(* Logix 5000 project; controller Project1Template vendor 1 type 14 code 151 rev 33.12; software revision 33.01; part 2 of 2 *)
(* tags used below, declared in another part *)
   SIM_ClampA : AOI_SIM_2PosCyl_ExtRet;
   SIM_ClampB : AOI_SIM_2PosCyl_ExtRet;
   SIM_ClampC : AOI_SIM_2PosCyl_ExtRet;
   SIM_EmptyFixture : TIMER;
   SIM_Fasten1 : AOI_SIM_RandomDelay;
   SIM_Fasten2 : AOI_SIM_RandomDelay;
   SIM_Fasten3 : AOI_SIM_RandomDelay;
   SIM_Fasten4 : AOI_SIM_RandomDelay;
   SIM_Fixture : AOI_SIM_2PosCyl_ExtRet;
   SIM_LightCurtainPartPlace : AOI_SIM_RandomDelay;
   SIM_LightCurtainPartRem : AOI_SIM_RandomDelay;
   SIM_NOP : BOOL;
   SIM_Oneshots : DINT;
   SIM_OperatorWorking : AOI_SIM_RandomDelay;
   SIM_PP_OFF : AOI_SIM_RandomDelay;
   SIM_PPA_ON : AOI_SIM_RandomDelay;
   SIM_PPB_ON : AOI_SIM_RandomDelay;
   SIM_PPC_ON : AOI_SIM_RandomDelay;
   SIM_PPD_ON : AOI_SIM_RandomDelay;
   SIM_RobotClear : AOI_SIM_RandomDelay;
   SIM_Torque : AOI_SIMAnalogSensor;
   F1_PASS : COUNTER;
   F2_PASS : COUNTER;
   F3_PASS : COUNTER;
   F4_PASS : COUNTER;
   FASTEN_AllComplete : BOOL;
   FASTEN_AllTorquesFail : BOOL;
   FASTEN_AllTorquesPass : BOOL;
   FASTEN_F1Complete : BOOL;
   FASTEN_F1Complete_ONS : BOOL;
   FASTEN_F1Torque : REAL;
   FASTEN_F1TorqueFail : BOOL;
   FASTEN_F1TorquePass : BOOL;
   FASTEN_F2Complete : BOOL;
   FASTEN_F2Complete_ONS : BOOL;
   FASTEN_F2Torque : REAL;
   FASTEN_F2TorqueFail : BOOL;
   FASTEN_F2TorquePass : BOOL;
   FASTEN_F3Complete : BOOL;
   FASTEN_F3Complete_ONS : BOOL;
   FASTEN_F3Torque : REAL;
   FASTEN_F3TorqueFail : BOOL;
   FASTEN_F3TorquePass : BOOL;
   FASTEN_F4Complete : BOOL;
   FASTEN_F4Complete_ONS : BOOL;
   FASTEN_F4Torque : REAL;
   FASTEN_F4TorqueFail : BOOL;
   FASTEN_F4TorquePass : BOOL;
   FASTEN_TorqueFeedback : REAL;
   FAULTS : DINT;
   FIXTURE_AllPartsPresent : BOOL;
   FIXTURE_AtHomePos : BOOL;
   FIXTURE_Empty : BOOL;
   FIXTURE_PartsSecured : BOOL;
   FIXTURE_PartsSecuredTmr : TIMER;
   FromHMI_ExtClampA_PB : BOOL;
   FromHMI_ExtClampB_PB : BOOL;
   FromHMI_ExtClampC_PB : BOOL;
   FromHMI_ExtFixture_PB : BOOL;
   FromHMI_F1LowLim : REAL;
   FromHMI_F1UppLim : REAL;
   FromHMI_F2LowLim : REAL;
   FromHMI_F2UppLim : REAL;
   FromHMI_F3LowLim : REAL;
   FromHMI_F3UppLim : REAL;
   FromHMI_F4LowLim : REAL;
   FromHMI_F4UppLim : REAL;
   FromHMI_RetClampA_PB : BOOL;
   FromHMI_RetClampB_PB : BOOL;
   FromHMI_RetClampC_PB : BOOL;
   FromHMI_RetFixture_PB : BOOL;
   FromHMI_StartPB : BOOL;
   FromHMI_StopPB : BOOL;
   FromRbt_ClearOfFixture : BOOL;
   FromRbt_Fasten1Complete : BOOL;
   FromRbt_Fasten2Complete : BOOL;
   FromRbt_Fasten3Complete : BOOL;
   FromRbt_Fasten4Complete : BOOL;
   HomePB : BOOL;
   I1 : INT;
   I2_CHA : REAL;   // Torque Sensor Input
   O3 : INT;
   SYS_AutoModeActive : BOOL;
   SYS_CycleActive : BOOL;
   SYS_ManualModeActive : BOOL;
   SYS_StartPBPulseTmr : TIMER;
   TIME : REAL;
   ToRbt_Fasten1Start : BOOL;
   ToRbt_Fasten2Start : BOOL;
   ToRbt_Fasten3Start : BOOL;
   ToRbt_Fasten4Start : BOOL;
(* MainProgram, continued *)

ROUTINE MainRoutine   (* ladder *)
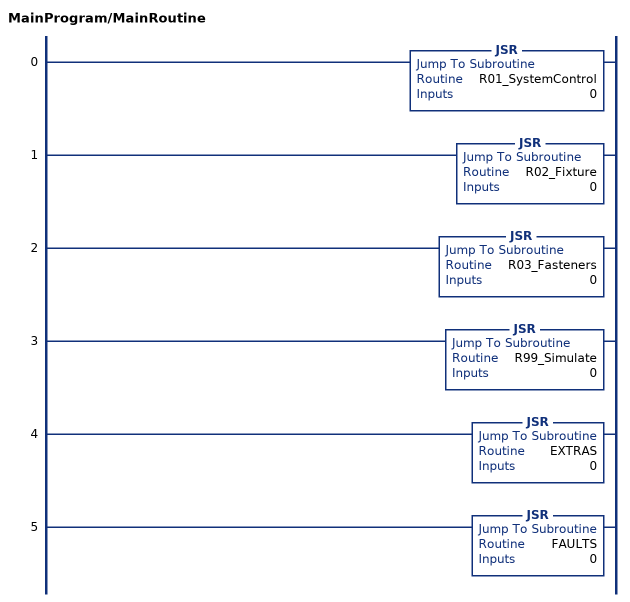
   0: JSR(R01_SystemControl,0);
   1: JSR(R02_Fixture,0);
   2: JSR(R03_Fasteners,0);
   3: JSR(R99_Simulate,0);
   4: JSR(EXTRAS,0);
   5: JSR(FAULTS,0);
END_ROUTINE

ROUTINE R01_SystemControl   (* ladder *)
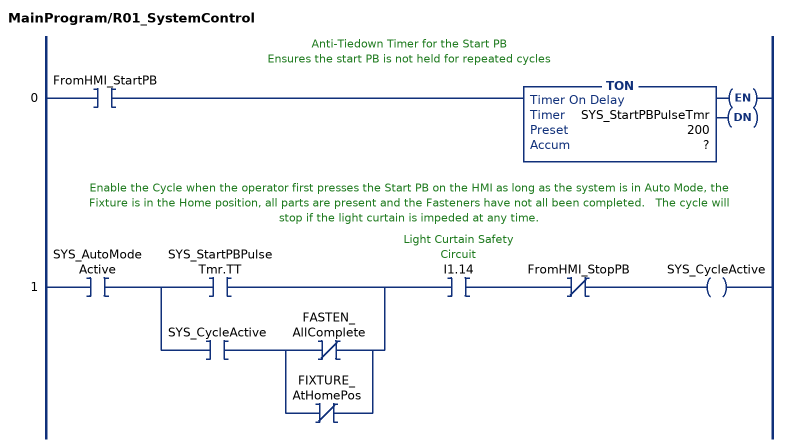
   // Anti-Tiedown Timer for the Start PB
   // Ensures the start PB is not held for repeated cycles
   0: XIC(FromHMI_StartPB)TON(SYS_StartPBPulseTmr,?,?);
   // Enable the Cycle when the operator first presses the Start PB on the HMI as long as the system is in Auto Mode, the Fixture is in the Home position, all parts are present and the Fasteners have not all been completed.   The cycle will stop if the light curtain is impeded at any time.
   1: XIC(SYS_AutoModeActive)[XIC(SYS_StartPBPulseTmr.TT) ,XIC(SYS_CycleActive) [XIO(FASTEN_AllComplete) ,XIO(FIXTURE_AtHomePos) ] ]XIC(I1.14)XIO(FromHMI_StopPB)OTE(SYS_CycleActive);
END_ROUTINE

ROUTINE R02_Fixture   (* ladder *)
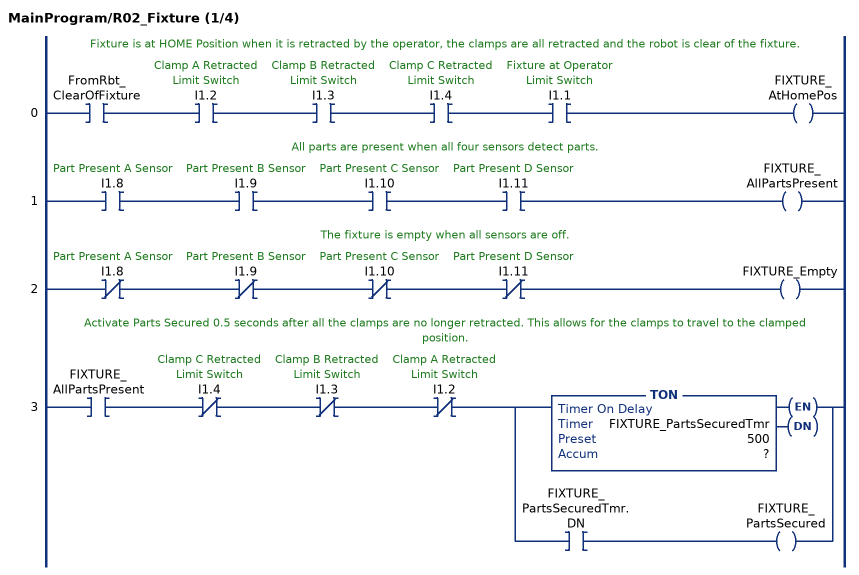
   // Fixture is at HOME Position when it is retracted by the operator, the clamps are all retracted and the robot is clear of the fixture.
   0: XIC(FromRbt_ClearOfFixture)XIC(I1.2)XIC(I1.3)XIC(I1.4)XIC(I1.1)OTE(FIXTURE_AtHomePos);
   // All parts are present when all four sensors detect parts.
   1: XIC(I1.8)XIC(I1.9)XIC(I1.10)XIC(I1.11)OTE(FIXTURE_AllPartsPresent);
   // The fixture is empty when all sensors are off.
   2: XIO(I1.8)XIO(I1.9)XIO(I1.10)XIO(I1.11)OTE(FIXTURE_Empty);
   // Activate Parts Secured 0.5 seconds after all the clamps are no longer retracted. This allows for the clamps to travel to the clamped position.
   3: XIC(FIXTURE_AllPartsPresent)XIO(I1.4)XIO(I1.3)XIO(I1.2)[TON(FIXTURE_PartsSecuredTmr,?,?) ,XIC(FIXTURE_PartsSecuredTmr.DN) OTE(FIXTURE_PartsSecured) ];
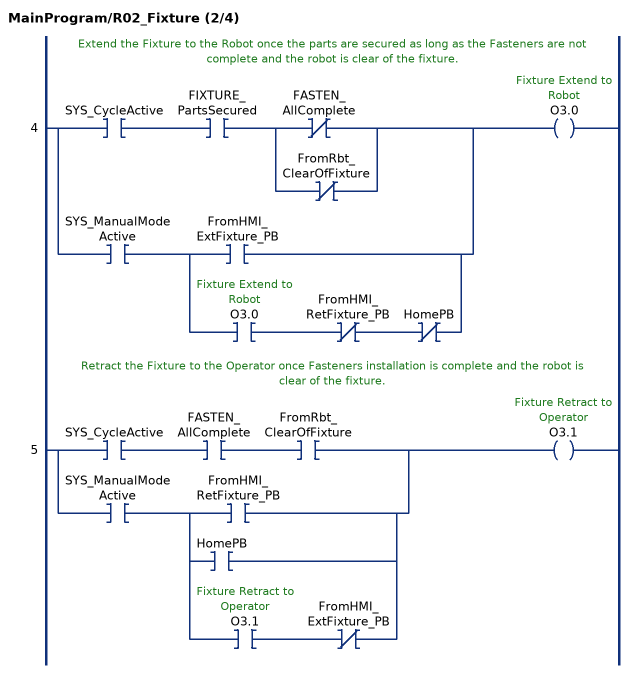
   // Extend the Fixture to the Robot once the parts are secured as long as the Fasteners are not complete and the robot is clear of the fixture.
   4: [XIC(SYS_CycleActive) XIC(FIXTURE_PartsSecured) [XIO(FASTEN_AllComplete) ,XIO(FromRbt_ClearOfFixture) ] ,XIC(SYS_ManualModeActive) [XIC(FromHMI_ExtFixture_PB) ,XIC(O3.0) XIO(FromHMI_RetFixture_PB) XIO(HomePB) ] ]OTE(O3.0);
   // Retract the Fixture to the Operator once Fasteners installation is complete and the robot is clear of the fixture.
   5: [XIC(SYS_CycleActive) XIC(FASTEN_AllComplete) XIC(FromRbt_ClearOfFixture) ,XIC(SYS_ManualModeActive) [[XIC(FromHMI_RetFixture_PB) ,XIC(HomePB) ] ,XIC(O3.1) XIO(FromHMI_ExtFixture_PB) ] ]OTE(O3.1);
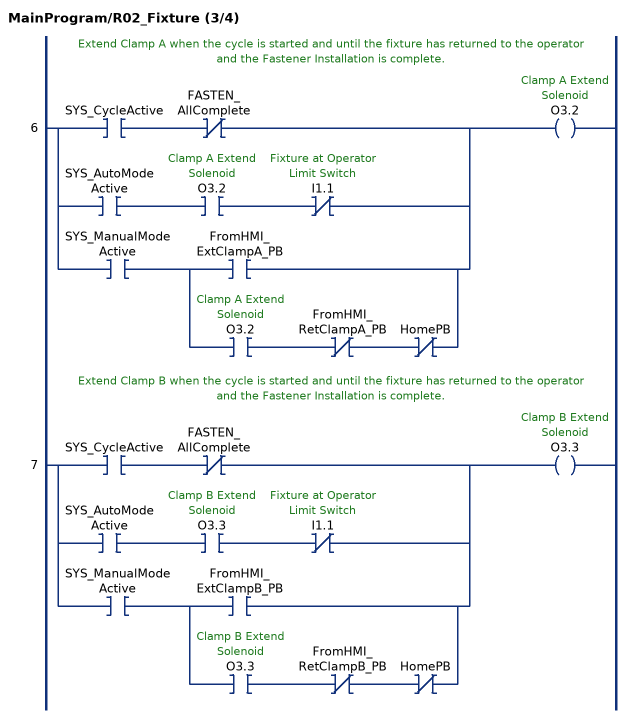
   // Extend Clamp A when the cycle is started and until the fixture has returned to the operator and the Fastener Installation is complete.
   6: [XIC(SYS_CycleActive) XIO(FASTEN_AllComplete) ,XIC(SYS_AutoModeActive) XIC(O3.2) XIO(I1.1) ,XIC(SYS_ManualModeActive) [XIC(FromHMI_ExtClampA_PB) ,XIC(O3.2) XIO(FromHMI_RetClampA_PB) XIO(HomePB) ] ]OTE(O3.2);
   // Extend Clamp B when the cycle is started and until the fixture has returned to the operator and the Fastener Installation is complete.
   7: [XIC(SYS_CycleActive) XIO(FASTEN_AllComplete) ,XIC(SYS_AutoModeActive) XIC(O3.3) XIO(I1.1) ,XIC(SYS_ManualModeActive) [XIC(FromHMI_ExtClampB_PB) ,XIC(O3.3) XIO(FromHMI_RetClampB_PB) XIO(HomePB) ] ]OTE(O3.3);
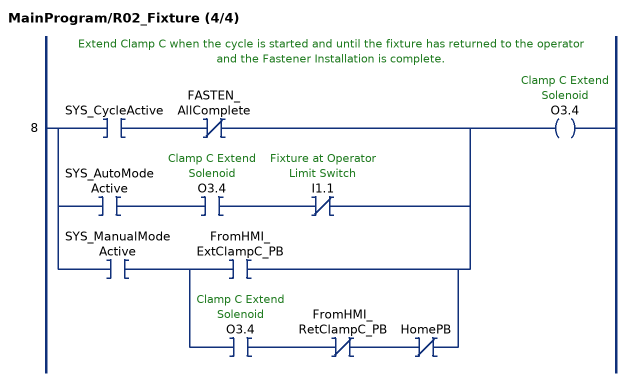
   // Extend Clamp C when the cycle is started and until the fixture has returned to the operator and the Fastener Installation is complete.
   8: [XIC(SYS_CycleActive) XIO(FASTEN_AllComplete) ,XIC(SYS_AutoModeActive) XIC(O3.4) XIO(I1.1) ,XIC(SYS_ManualModeActive) [XIC(FromHMI_ExtClampC_PB) ,XIC(O3.4) XIO(FromHMI_RetClampC_PB) XIO(HomePB) ] ]OTE(O3.4);
END_ROUTINE

ROUTINE R03_Fasteners   (* ladder *)
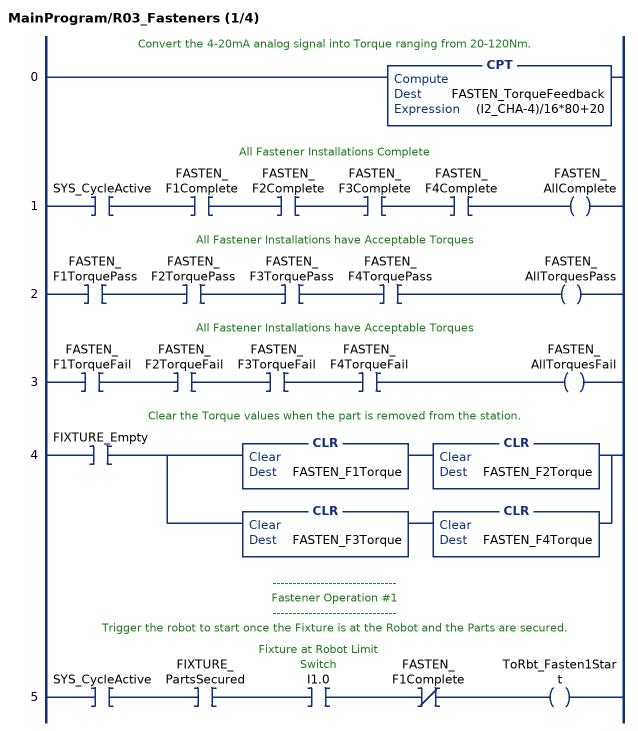
   // Convert the 4-20mA analog signal into Torque ranging from 20-120Nm.
   0: CPT(FASTEN_TorqueFeedback,(I2_CHA-4)/16*80+20);
   // All Fastener Installations Complete
   1: XIC(SYS_CycleActive)XIC(FASTEN_F1Complete)XIC(FASTEN_F2Complete)XIC(FASTEN_F3Complete)XIC(FASTEN_F4Complete)OTE(FASTEN_AllComplete);
   // All Fastener Installations have Acceptable Torques
   2: XIC(FASTEN_F1TorquePass)XIC(FASTEN_F2TorquePass)XIC(FASTEN_F3TorquePass)XIC(FASTEN_F4TorquePass)OTE(FASTEN_AllTorquesPass);
   // All Fastener Installations have Acceptable Torques
   3: XIC(FASTEN_F1TorqueFail)XIC(FASTEN_F2TorqueFail)XIC(FASTEN_F3TorqueFail)XIC(FASTEN_F4TorqueFail)OTE(FASTEN_AllTorquesFail);
   // Clear the Torque values when the part is removed from the station.
   4: XIC(FIXTURE_Empty)[CLR(FASTEN_F1Torque) CLR(FASTEN_F2Torque) ,CLR(FASTEN_F3Torque) CLR(FASTEN_F4Torque) ];
   // -------------------------------
   // Fastener Operation #1
   // -------------------------------
   // Trigger the robot to start once the Fixture is at the Robot and the Parts are secured.
   5: XIC(SYS_CycleActive)XIC(FIXTURE_PartsSecured)XIC(I1.0)XIO(FASTEN_F1Complete)OTE(ToRbt_Fasten1Start);
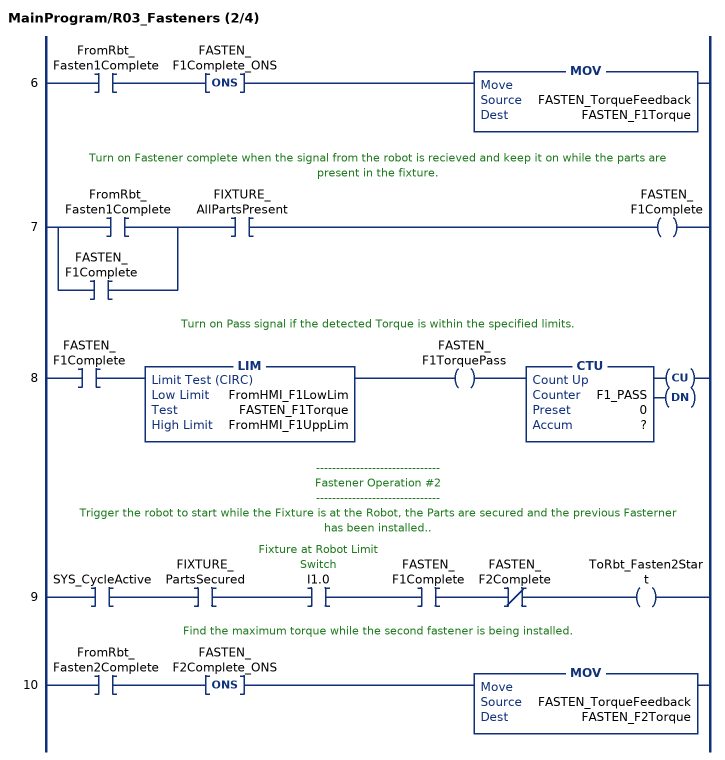
   6: XIC(FromRbt_Fasten1Complete)ONS(FASTEN_F1Complete_ONS)MOV(FASTEN_TorqueFeedback,FASTEN_F1Torque);
   // Turn on Fastener complete when the signal from the robot is recieved and keep it on while the parts are present in the fixture.
   7: [XIC(FromRbt_Fasten1Complete) ,XIC(FASTEN_F1Complete) ]XIC(FIXTURE_AllPartsPresent)OTE(FASTEN_F1Complete);
   // Turn on Pass signal if the detected Torque is within the specified limits.
   8: XIC(FASTEN_F1Complete)LIM(FromHMI_F1LowLim,FASTEN_F1Torque,FromHMI_F1UppLim)OTE(FASTEN_F1TorquePass)CTU(F1_PASS,?,?);
   // -------------------------------
   // Fastener Operation #2
   // -------------------------------
   // Trigger the robot to start while the Fixture is at the Robot, the Parts are secured and the previous Fasterner has been installed..
   9: XIC(SYS_CycleActive)XIC(FIXTURE_PartsSecured)XIC(I1.0)XIC(FASTEN_F1Complete)XIO(FASTEN_F2Complete)OTE(ToRbt_Fasten2Start);
   // Find the maximum torque while the second fastener is being installed.
   10: XIC(FromRbt_Fasten2Complete)ONS(FASTEN_F2Complete_ONS)MOV(FASTEN_TorqueFeedback,FASTEN_F2Torque);
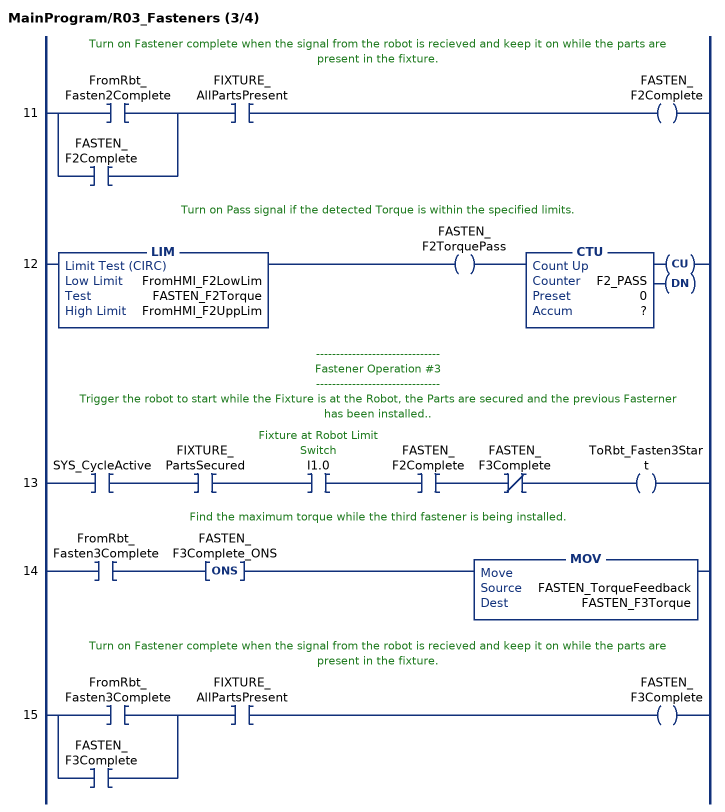
   // Turn on Fastener complete when the signal from the robot is recieved and keep it on while the parts are present in the fixture.
   11: [XIC(FromRbt_Fasten2Complete) ,XIC(FASTEN_F2Complete) ]XIC(FIXTURE_AllPartsPresent)OTE(FASTEN_F2Complete);
   // Turn on Pass signal if the detected Torque is within the specified limits.
   12: LIM(FromHMI_F2LowLim,FASTEN_F2Torque,FromHMI_F2UppLim)OTE(FASTEN_F2TorquePass)CTU(F2_PASS,?,?);
   // -------------------------------
   // Fastener Operation #3
   // -------------------------------
   // Trigger the robot to start while the Fixture is at the Robot, the Parts are secured and the previous Fasterner has been installed..
   13: XIC(SYS_CycleActive)XIC(FIXTURE_PartsSecured)XIC(I1.0)XIC(FASTEN_F2Complete)XIO(FASTEN_F3Complete)OTE(ToRbt_Fasten3Start);
   // Find the maximum torque while the third fastener is being installed.
   14: XIC(FromRbt_Fasten3Complete)ONS(FASTEN_F3Complete_ONS)MOV(FASTEN_TorqueFeedback,FASTEN_F3Torque);
   // Turn on Fastener complete when the signal from the robot is recieved and keep it on while the parts are present in the fixture.
   15: [XIC(FromRbt_Fasten3Complete) ,XIC(FASTEN_F3Complete) ]XIC(FIXTURE_AllPartsPresent)OTE(FASTEN_F3Complete);
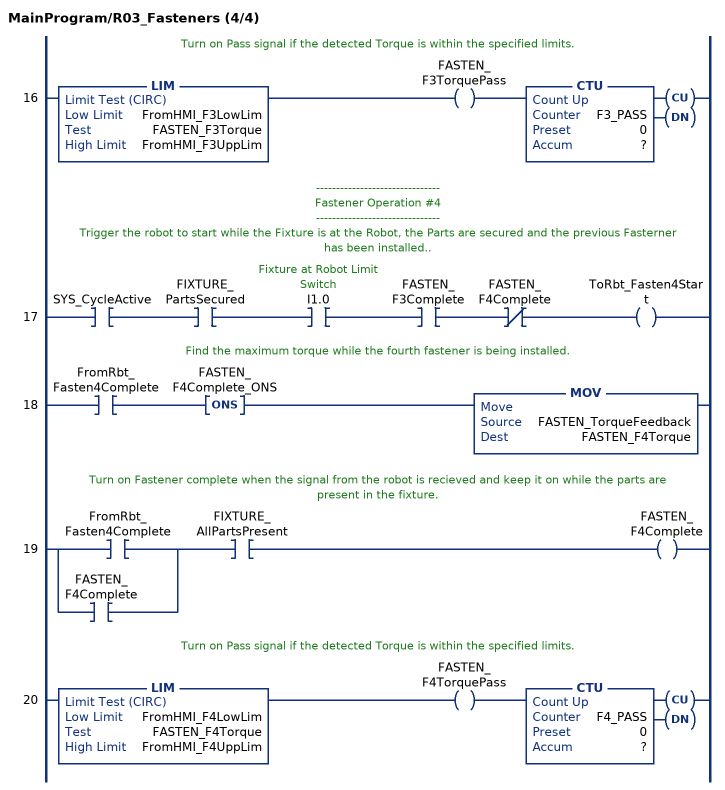
   // Turn on Pass signal if the detected Torque is within the specified limits.
   16: LIM(FromHMI_F3LowLim,FASTEN_F3Torque,FromHMI_F3UppLim)OTE(FASTEN_F3TorquePass)CTU(F3_PASS,?,?);
   // -------------------------------
   // Fastener Operation #4
   // -------------------------------
   // Trigger the robot to start while the Fixture is at the Robot, the Parts are secured and the previous Fasterner has been installed..
   17: XIC(SYS_CycleActive)XIC(FIXTURE_PartsSecured)XIC(I1.0)XIC(FASTEN_F3Complete)XIO(FASTEN_F4Complete)OTE(ToRbt_Fasten4Start);
   // Find the maximum torque while the fourth fastener is being installed.
   18: XIC(FromRbt_Fasten4Complete)ONS(FASTEN_F4Complete_ONS)MOV(FASTEN_TorqueFeedback,FASTEN_F4Torque);
   // Turn on Fastener complete when the signal from the robot is recieved and keep it on while the parts are present in the fixture.
   19: [XIC(FromRbt_Fasten4Complete) ,XIC(FASTEN_F4Complete) ]XIC(FIXTURE_AllPartsPresent)OTE(FASTEN_F4Complete);
   // Turn on Pass signal if the detected Torque is within the specified limits.
   20: LIM(FromHMI_F4LowLim,FASTEN_F4Torque,FromHMI_F4UppLim)OTE(FASTEN_F4TorquePass)CTU(F4_PASS,?,?);
END_ROUTINE

ROUTINE R98_DemoMonitoring   (* ladder *)
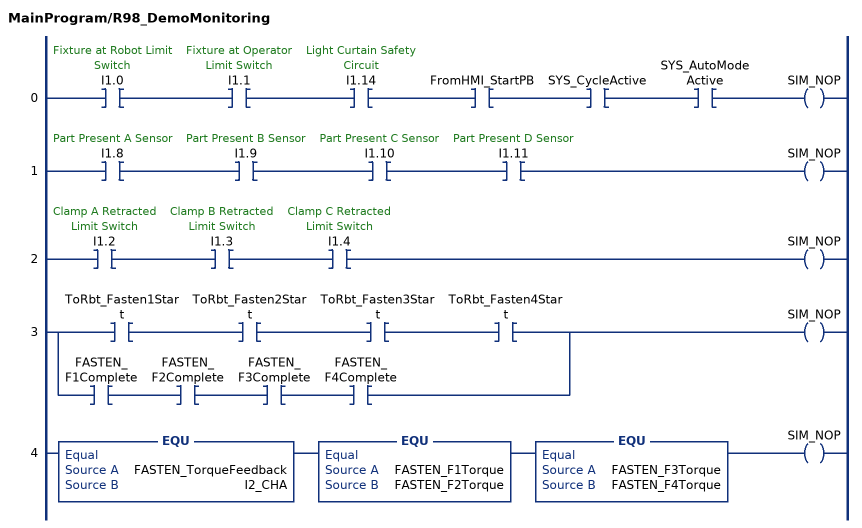
   0: XIC(I1.0)XIC(I1.1)XIC(I1.14)XIC(FromHMI_StartPB)XIC(SYS_CycleActive)XIC(SYS_AutoModeActive)OTE(SIM_NOP);
   1: XIC(I1.8)XIC(I1.9)XIC(I1.10)XIC(I1.11)OTE(SIM_NOP);
   2: XIC(I1.2)XIC(I1.3)XIC(I1.4)OTE(SIM_NOP);
   3: [XIC(ToRbt_Fasten1Start) XIC(ToRbt_Fasten2Start) XIC(ToRbt_Fasten3Start) XIC(ToRbt_Fasten4Start) ,XIC(FASTEN_F1Complete) XIC(FASTEN_F2Complete) XIC(FASTEN_F3Complete) XIC(FASTEN_F4Complete) ]OTE(SIM_NOP);
   4: EQU(FASTEN_TorqueFeedback,I2_CHA)EQU(FASTEN_F1Torque,FASTEN_F2Torque)EQU(FASTEN_F3Torque,FASTEN_F4Torque)OTE(SIM_NOP);
END_ROUTINE

ROUTINE R99_Simulate   (* ladder *)
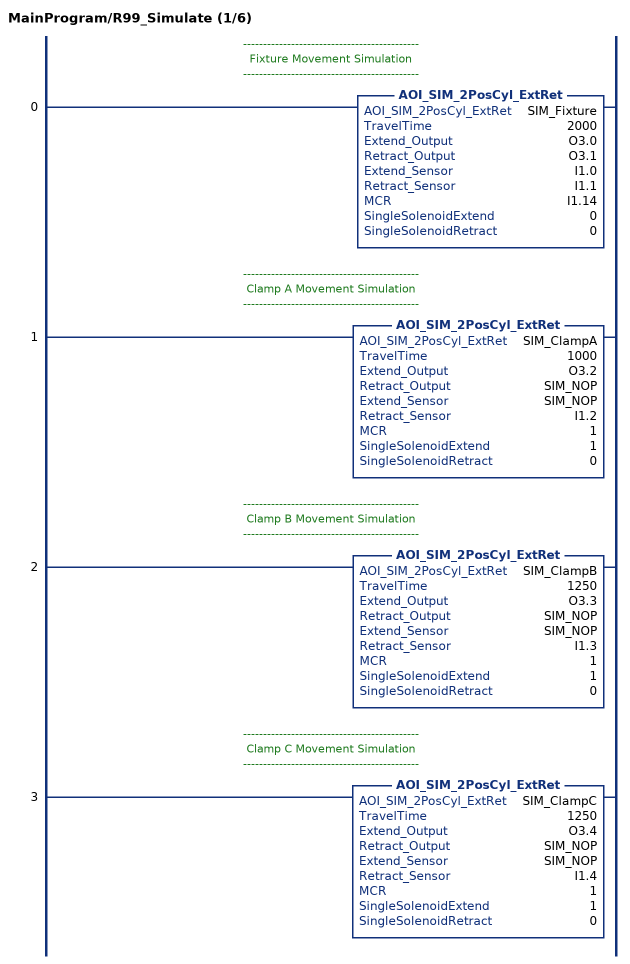
   // --------------------------------------------
   // Fixture Movement Simulation
   // --------------------------------------------
   0: AOI_SIM_2PosCyl_ExtRet(SIM_Fixture,2000,O3.0,O3.1,I1.0,I1.1,I1.14,0,0);
   // --------------------------------------------
   // Clamp A Movement Simulation
   // --------------------------------------------
   1: AOI_SIM_2PosCyl_ExtRet(SIM_ClampA,1000,O3.2,SIM_NOP,SIM_NOP,I1.2,1,1,0);
   // --------------------------------------------
   // Clamp B Movement Simulation
   // --------------------------------------------
   2: AOI_SIM_2PosCyl_ExtRet(SIM_ClampB,1250,O3.3,SIM_NOP,SIM_NOP,I1.3,1,1,0);
   // --------------------------------------------
   // Clamp C Movement Simulation
   // --------------------------------------------
   3: AOI_SIM_2PosCyl_ExtRet(SIM_ClampC,1250,O3.4,SIM_NOP,SIM_NOP,I1.4,1,1,0);
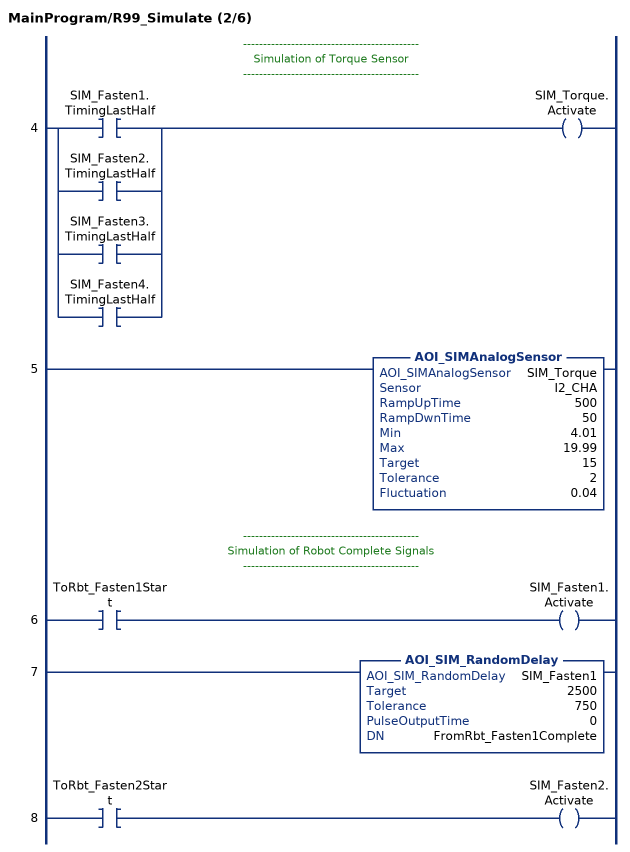
   // --------------------------------------------
   // Simulation of Torque Sensor
   // --------------------------------------------
   4: [XIC(SIM_Fasten1.TimingLastHalf) ,XIC(SIM_Fasten2.TimingLastHalf) ,XIC(SIM_Fasten3.TimingLastHalf) ,XIC(SIM_Fasten4.TimingLastHalf) ]OTE(SIM_Torque.Activate);
   5: AOI_SIMAnalogSensor(SIM_Torque,I2_CHA,500,50,4.01,19.99,15,2,0.04);
   // --------------------------------------------
   // Simulation of Robot Complete Signals
   // --------------------------------------------
   6: XIC(ToRbt_Fasten1Start)OTE(SIM_Fasten1.Activate);
   7: AOI_SIM_RandomDelay(SIM_Fasten1,2500,750,0,FromRbt_Fasten1Complete);
   8: XIC(ToRbt_Fasten2Start)OTE(SIM_Fasten2.Activate);
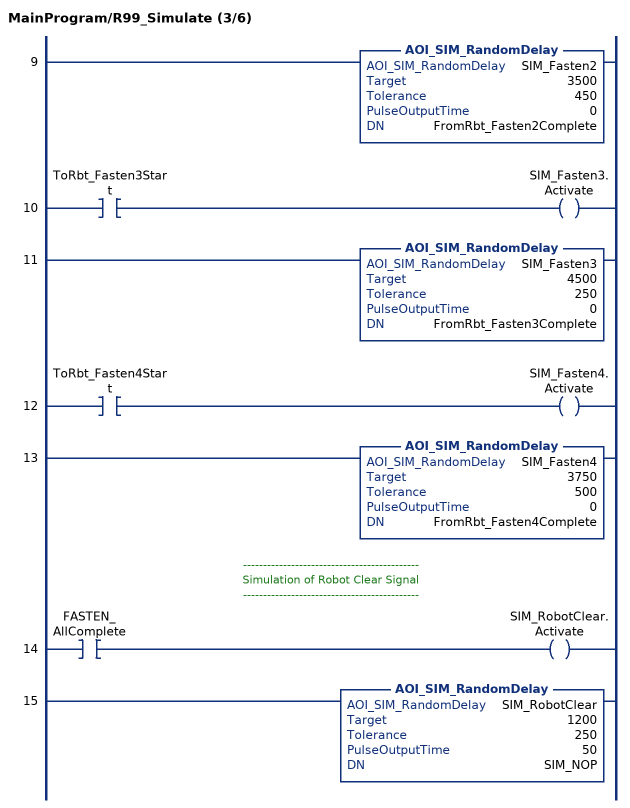
   9: AOI_SIM_RandomDelay(SIM_Fasten2,3500,450,0,FromRbt_Fasten2Complete);
   10: XIC(ToRbt_Fasten3Start)OTE(SIM_Fasten3.Activate);
   11: AOI_SIM_RandomDelay(SIM_Fasten3,4500,250,0,FromRbt_Fasten3Complete);
   12: XIC(ToRbt_Fasten4Start)OTE(SIM_Fasten4.Activate);
   13: AOI_SIM_RandomDelay(SIM_Fasten4,3750,500,0,FromRbt_Fasten4Complete);
   // --------------------------------------------
   // Simulation of Robot Clear Signal
   // --------------------------------------------
   14: XIC(FASTEN_AllComplete)OTE(SIM_RobotClear.Activate);
   15: AOI_SIM_RandomDelay(SIM_RobotClear,1200,250,50,SIM_NOP);
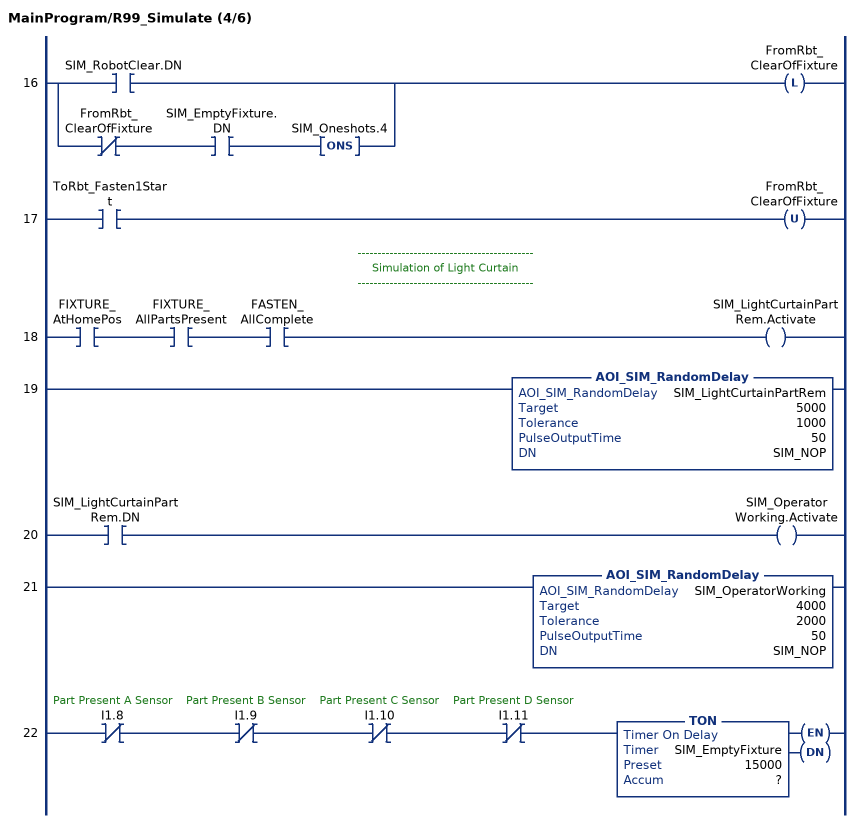
   16: [XIC(SIM_RobotClear.DN) ,XIO(FromRbt_ClearOfFixture) XIC(SIM_EmptyFixture.DN) ONS(SIM_Oneshots.4) ]OTL(FromRbt_ClearOfFixture);
   17: XIC(ToRbt_Fasten1Start)OTU(FromRbt_ClearOfFixture);
   // --------------------------------------------
   // Simulation of Light Curtain
   // --------------------------------------------
   18: XIC(FIXTURE_AtHomePos)XIC(FIXTURE_AllPartsPresent)XIC(FASTEN_AllComplete)OTE(SIM_LightCurtainPartRem.Activate);
   19: AOI_SIM_RandomDelay(SIM_LightCurtainPartRem,5000,1000,50,SIM_NOP);
   20: XIC(SIM_LightCurtainPartRem.DN)OTE(SIM_OperatorWorking.Activate);
   21: AOI_SIM_RandomDelay(SIM_OperatorWorking,4000,2000,50,SIM_NOP);
   22: XIO(I1.8)XIO(I1.9)XIO(I1.10)XIO(I1.11)TON(SIM_EmptyFixture,?,?);
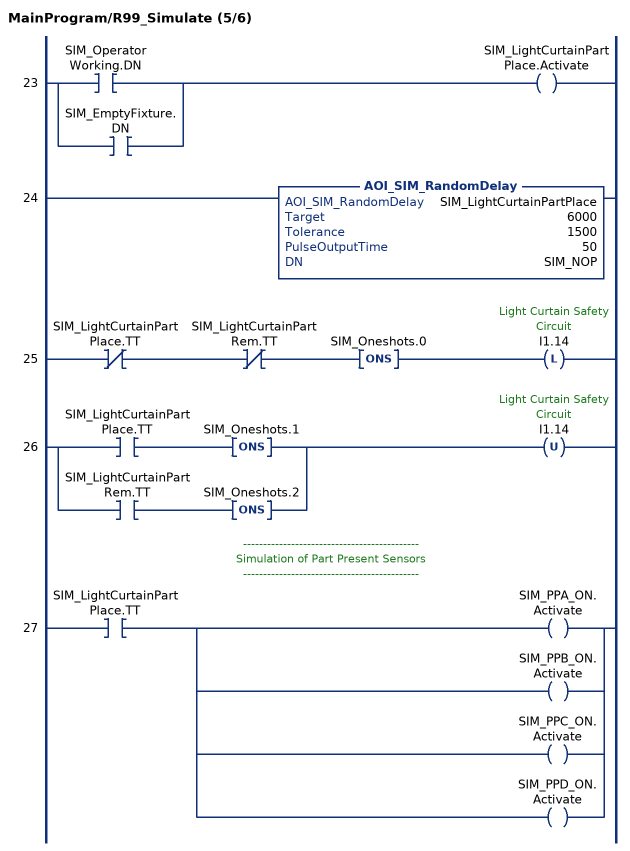
   23: [XIC(SIM_OperatorWorking.DN) ,XIC(SIM_EmptyFixture.DN) ]OTE(SIM_LightCurtainPartPlace.Activate);
   24: AOI_SIM_RandomDelay(SIM_LightCurtainPartPlace,6000,1500,50,SIM_NOP);
   25: XIO(SIM_LightCurtainPartPlace.TT)XIO(SIM_LightCurtainPartRem.TT)ONS(SIM_Oneshots.0)OTL(I1.14);
   26: [XIC(SIM_LightCurtainPartPlace.TT) ONS(SIM_Oneshots.1) ,XIC(SIM_LightCurtainPartRem.TT) ONS(SIM_Oneshots.2) ]OTU(I1.14);
   // --------------------------------------------
   // Simulation of Part Present Sensors
   // --------------------------------------------
   27: XIC(SIM_LightCurtainPartPlace.TT)[OTE(SIM_PPA_ON.Activate) ,OTE(SIM_PPB_ON.Activate) ,OTE(SIM_PPC_ON.Activate) ,OTE(SIM_PPD_ON.Activate) ];
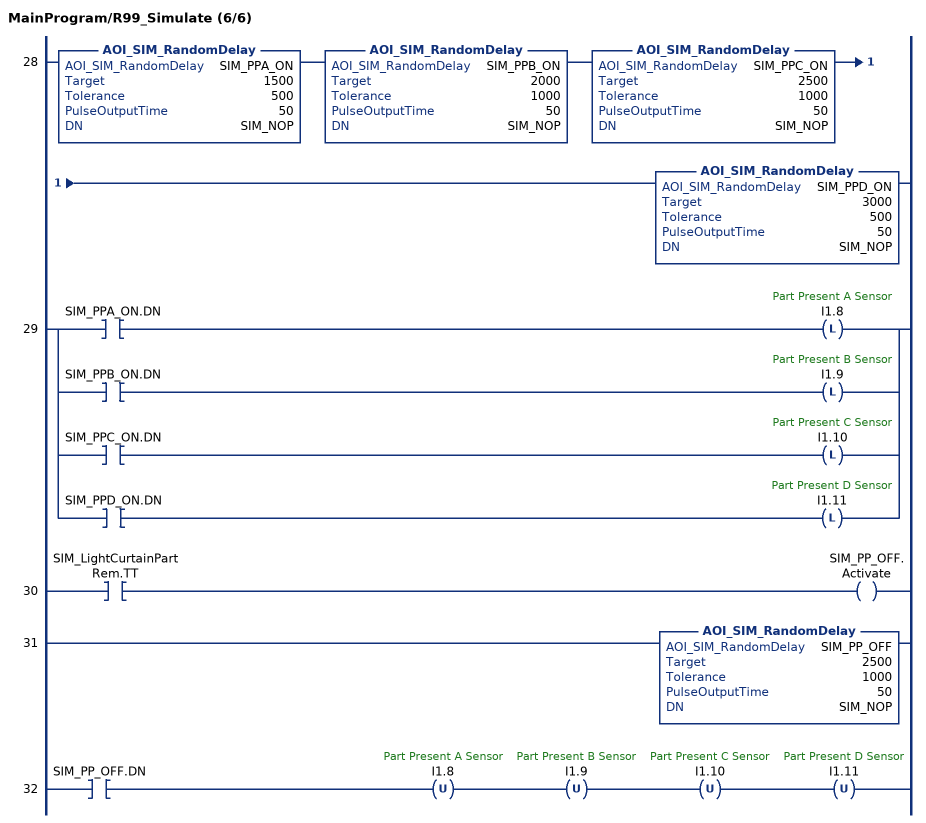
   28: AOI_SIM_RandomDelay(SIM_PPA_ON,1500,500,50,SIM_NOP)AOI_SIM_RandomDelay(SIM_PPB_ON,2000,1000,50,SIM_NOP)AOI_SIM_RandomDelay(SIM_PPC_ON,2500,1000,50,SIM_NOP)AOI_SIM_RandomDelay(SIM_PPD_ON,3000,500,50,SIM_NOP);
   29: [XIC(SIM_PPA_ON.DN) OTL(I1.8) ,XIC(SIM_PPB_ON.DN) OTL(I1.9) ,XIC(SIM_PPC_ON.DN) OTL(I1.10) ,XIC(SIM_PPD_ON.DN) OTL(I1.11) ];
   30: XIC(SIM_LightCurtainPartRem.TT)OTE(SIM_PP_OFF.Activate);
   31: AOI_SIM_RandomDelay(SIM_PP_OFF,2500,1000,50,SIM_NOP);
   32: XIC(SIM_PP_OFF.DN)OTU(I1.8)OTU(I1.9)OTU(I1.10)OTU(I1.11);
END_ROUTINE
END_PROGRAM
